RoboDK station: Station (1) — копия — копия.rdk

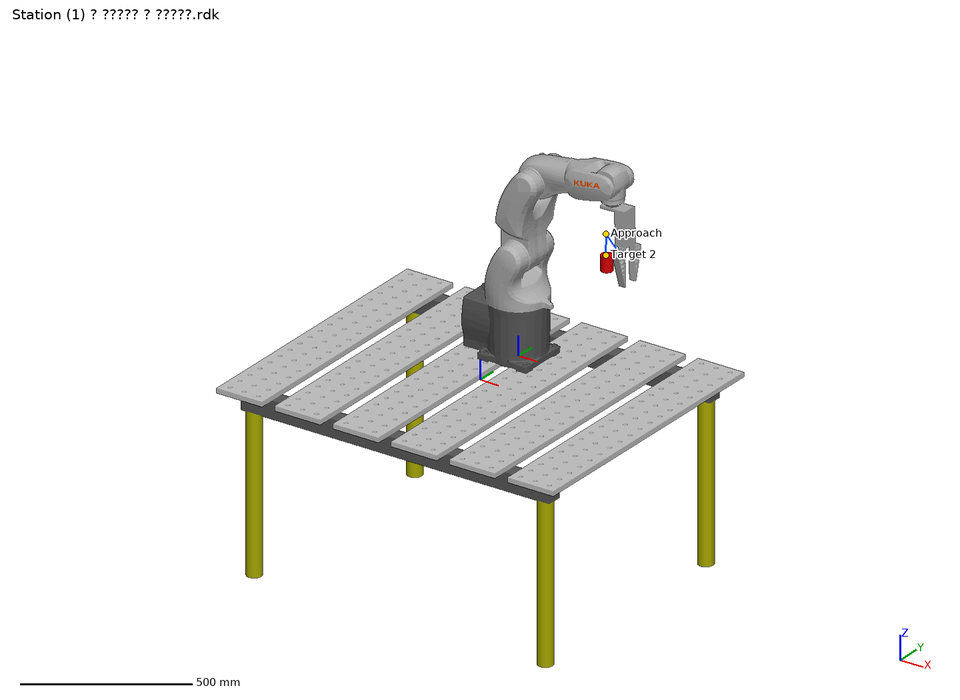
[picture v0: the station drawn from its stored meshes, robots at their saved joint values, targets as dots, program paths as lines]
Station Station (1). Poses are relative to the parent item; angles as X-Y-Z fixed-axis rotations.
  - frame KUKA KR 3 R540 Base at (0, 199.71, 0) mm
    - robot KUKA KR 3 R540: 6 axes, payload 3 kg, reach 541 mm, repeatability 0.02 mm, weight 26 kg
        modified DH rows (alpha deg, a mm, theta deg, d mm): 0, 0, 0, 345; -90, 20, 0, 0; 0, 260, -90, 0; -90, 20, 0, 260; 90, 0, 0, 0; -90, 0, 180, 75
        joint limits [-170, -170, -110, -175, -120, -350] to [170, 50, 155, 175, 120, 350]; home [0, -90, 90, 0, 0, 0]; saved at [0, -77.419, 69.671, 0, 96.213, 0]
      - tool Gripper Closed, TCP at (-40, 0, 200) mm, size 87.7 x 99.2 x 241.1 mm, geometry from c2.stl
      - tool Gripper Opened, TCP at (-40, 0, 200) mm, size 87.7 x 115.5 x 241.4 mm, geometry from case opened v2.stl
    - target Approach (Cartesian target) at (236.76, 105.25, 417.17) mm, rotated rx -180 ry 0.76 rz -180 deg; joints [-28.592, -99.885, 83.982, 0.377, 105.236, -28.49] of KUKA KR 3 R540
    - target Target 2 (Cartesian target) at (249.53, 85.6, 360.32) mm, rotated rx 180 ry 0.76 rz -180 deg; joints [-22.575, -102.29, 98.815, 0.292, 92.773, -22.559] of KUKA KR 3 R540
    - target Target 3 (Cartesian target) at (262.05, 142.05, 342.29) mm, rotated rx 180 ry 0.76 rz -180 deg; joints [-33.039, -94.397, 96.048, 0.415, 87.711, -33.054] of KUKA KR 3 R540
  - program Prog1 (16 instructions, listed below)
  - frame Frame 2 at (0, 4.53, 0) mm
    - object Table at (0, 0, 0) mm, size 1193.8 x 965.2 x 609.6 mm, geometry from welding_table.sld
  - program Replace objects (1 instructions, listed below)
  - Python program Смыкание и размыкание клешни (listed below)
  - object Part at (250.91, 287.96, 351.48) mm, size 37.8 x 37.8 x 50.4 mm, geometry from part.sld
  - program arman (10 instructions, listed below)
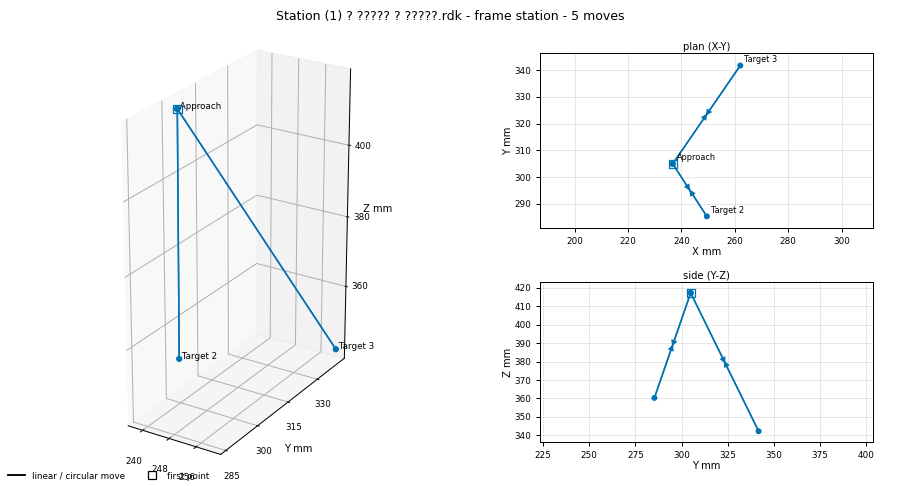
[picture p0: tool path of Station (1) — копия — копия.rdk in frame station, 5 of 5 moves have a stored position in this frame; points joined in program order, loops and branches not executed]

--- program Prog1 (robot KUKA KR 3 R540) ---
  Set speed (20.0 mm/s)
  Set Ref.: KUKA KR 3 R540 Base
  Set Tool: Gripper Closed
  MoveL (Approach)
  MoveL (Target 2)
  Pause 1.0 s
  Attach to Gripper Closed
  Pause 1.5 s
  Set Ref.: Frame 2
  MoveL (Approach)
  MoveL (Target 3)
  Pause 1.0 s
  Detach from Gripper Closed
  Pause 1.5 s
  MoveL (Approach)
  Call Replace objects

--- program Replace objects (robot KUKA KR 3 R540) ---
  Replace objects

--- Python program Смыкание и размыкание клешни ---
# Type help("robolink") or help("robodk") for more information
# Press F5 to run the script
# Note: you do not need to keep a copy of this file, your python script is saved with the station
from robolink import *    # API to communicate with RoboDK
from robodk import *      # basic matrix operations
RDK = Robolink()

# This file allows simulating the opening and closing of grippers.
# Two models of the gripper per robot are required: one opened and one closed.
# The opened model of the gripper should have the keyword "Opened"
# The closed model of the gripper should have the keyword "Closed"
# Simply place this file in the station and leave it running to
# make it work

OPENED_KEYWORD = 'Opened'
CLOSED_KEYWORD = 'Closed'
UPDATE_FREQUENCY = 0.01

# Loop forever
print('Starting infinite loop to simulate open/close of tools')
while True:
    # First step: get a list of tool pairs (open, closed) per robot
    Tool_Pairs = []
    # get all the robot names (strings)
    all_robots = RDK.ItemList(ITEM_TYPE_ROBOT, True)
    for i in range(len(all_robots)):
        roboti = RDK.Item(all_robots[i])
        roboti_name = roboti.Name()
        # get the tools of each robot
        roboti_tools = roboti.Childs()
        opened = None
        closed = None
        # store the opened model and closed model of each gripper
        for t in range(len(roboti_tools)):
            tnamei = roboti_tools[t].Name()
            if not isinstance(opened,Item) and tnamei.count(OPENED_KEYWORD) > 0:
                opened = roboti_tools[t]
                print('Using %s from robot %s as gripper opened' % (tnamei, roboti_name))
            elif not isinstance(closed,Item) and tnamei.count(CLOSED_KEYWORD) > 0:
                closed = roboti_tools[t]
                print('Using %s from robot %s as gripper closed' % (tnamei, roboti_name))

            if isinstance(opened, Item) and isinstance(closed, Item):
                # Stop if we have an open state and a closed state per robot
                break;
        Tool_Pairs.append([opened, closed])

    # We may find as many pairs of tools as robots are available in the station
    nTool_Pairs = len(Tool_Pairs)
    while True:
        #try:
                # Iterate through all tool pairs and detect the presence of objects
            for i in range(nTool_Pairs):
                opened = Tool_Pairs[i][0]
                closed = Tool_Pairs[i][1]
                open_valid = isinstance(opened,Item)
                close_valid = isinstance(closed,Item)
                tool_is_open = True

                # Check if the tool holds one or more objects:
                if (open_valid and len(opened.Childs()) > 0) or (close_valid and len(closed.Childs()) > 0):
                    tool_is_open = False

                # Update the visibility of the tools
                if open_valid:
                    opened.setVisible(tool_is_open)
                if close_valid:
                    closed.setVisible(not tool_is_open)

            # Take a pause...
            pause(UPDATE_FREQUENCY)

                #except:
                     #print('An item was deleted. Remaking tool list')
                #break

--- program arman (robot KUKA KR 3 R540) ---
  INI
  while TRUE
  OUT 1 'gripper_open' State=F...: OUT 1 'gripper_open' State=FALSE
  wait sec 1
  OUT 2 'gripper_close' State=...: OUT 2 'gripper_close' State=TRUE
  wait sec 1
  OUT 2 'gripper_close' State=...: OUT 2 'gripper_close' State=FALSE
  wait sec 1
  ENDWHILE
  END
